Fanuc KAREL source: NC0034.KL

-- PROVISIONAL review KL for V1013-1; original PC SHA256 a74cb3c65fad4d94fdcb64d8cb372f789559f63bae3181bfb92a775a752311d3
-- Incomplete behavior may be omitted. Consult companion uncertainty JSON. Do not deploy.
PROGRAM NC0034
%NOLOCKGROUP
-- UNRESOLVED_LOCAL_POOL 1 cells at code offset 3; source declarations unknown
-- DIRECT_LOCAL_WORD_ACCESS alone does not prove INTEGER, REAL, or BOOLEAN
BEGIN
  -- UNRESOLVED_PC offsets 0-8; opcodes 2B,2C,7B
  -- UNRESOLVED_PC offsets 13-20; opcodes 9D,23
  -- UNRESOLVED_PC offsets 25-42; opcodes 21,40,41,42
  -- UNRESOLVED_PC offsets 47-81; opcodes 21,2E,52,23,7A,40,41,42
  -- UNRESOLVED_PC offsets 86-110; opcodes 21,2E,52,23,7A,43
  -- UNRESOLVED_PC offsets 115-132; opcodes 21,40,41,42
  -- UNRESOLVED_PC offsets 137-171; opcodes 21,2E,52,23,7A,40,41,42
  -- UNRESOLVED_PC offsets 176-200; opcodes 21,2E,52,23,7A,43
  -- UNRESOLVED_PC offsets 205-222; opcodes 21,40,41,42
  -- UNRESOLVED_PC offsets 227-261; opcodes 21,2E,52,23,7A,40,41,42
  -- UNRESOLVED_PC offsets 266-290; opcodes 21,2E,52,23,7A,43
  -- UNRESOLVED_PC offsets 295-309; opcodes 21,9D,52,23
  -- UNRESOLVED_PC offsets 329-333; opcodes 7F
  -- UNRESOLVED_PC offsets 338-342; opcodes 27,AA
  -- UNRESOLVED_PC offsets 347-351; opcodes 7F
END NC0034
